TYPE
    IOAxis :
    STRUCT
        GateWayStatus  : GatewayStatus;
        GateWayControl : GatewayControl;
        PlcInFromAxis  : PlcIn;
        PlcOutToAxis   : PlcOut;
    END_STRUCT
END_TYPE

(* stored: Version 1.1.0.1, ProductVersion 3.1.4024.12
   DUT IOAxis: Id {a1b2396f-d4df-447a-ac59-9633d87627af} *)
